// This function has been automatically generated from the project information.
{attribute 'signature_flag' := '1073741824'}
{attribute 'TcGenerated'}
{attribute 'no-analysis'}
FUNCTION F_GetCompany : WSTRING
VAR_INPUT
	
END_VAR

F_GetCompany := "Sawtooth Robotics";

END_FUNCTION

(* stored: Version 1.1.0.1
   POU F_GetCompany: Id {0c788959-3d13-4c16-b4d8-186dc79f7eb8}, SpecialFunc None *)
